(*
A queryable interface designed for transmitting data via a `Broadcast` system.  
Allows debugging and querying.
*)
INTERFACE I_Arg EXTENDS __SYSTEM.IQueryInterface, I_Debug

END_INTERFACE

(* stored: Version 1.1.0.1
   Itf I_Arg: Id {e29f84e2-8703-4b76-ad19-a0ce9ce24d7a} *)
